FUNCTION_BLOCK GoToInit IMPLEMENTS I_Transitive
VAR
    _currentState : POINTER TO I_SD_ValveState;
    _nextState : REFERENCE TO InitState;
END_VAR

METHOD FB_init : BOOL
VAR_INPUT
	bInitRetains : BOOL; // if TRUE, the retain variables are initialized (warm start / cold start)
	bInCopyCode : BOOL;  // if TRUE, the instance afterwards gets moved into the copy code (online change)
    currentState : POINTER TO I_SD_ValveState;
    nextState : REFERENCE TO InitState;
END_VAR
_currentState := currentState;
_nextState REF= nextState;
END_METHOD

METHOD Transit
_currentState^ := _nextState;
END_METHOD

END_FUNCTION_BLOCK

(* stored: Version 1.1.0.1, ProductVersion 3.1.4024.12
   POU GoToInit: Id {b00b96b1-8aa0-4b43-9bcf-be88fc645a25}, SpecialFunc None
   Method FB_init: Id {81b97a08-793b-4446-a19e-6658f4842a75}
   Method Transit: Id {35919353-e761-4906-9cb8-4fe087149a02} *)
